FUNCTION_BLOCK E_SH_BYTE (* Sample-and-Hold for BOOL *)
  (* Standard: 61499-2 *)
  (* Version 1.0, 2024-02-23, franz *)
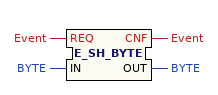
  EVENT_INPUT
    REQ; (* Normal Execution Request *)
  END_EVENT
  EVENT_OUTPUT
    CNF; (* Execution Confirmation *)
  END_EVENT
  VAR_INPUT
    IN : BYTE; (* Sample *)
  END_VAR
  VAR_OUTPUT
    OUT : BYTE; (* Hold *)
  END_VAR
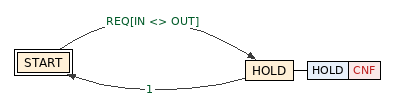
  EC_STATES
    START; (* Initial State *)
    HOLD : HOLD -> CNF;
  END_STATES
  EC_TRANSITIONS
    START TO HOLD := REQ[IN <> OUT];
    HOLD TO START := 1;
  END_TRANSITIONS
  ALGORITHM HOLD IN ST:
OUT := IN;
  END_ALGORITHM
END_FUNCTION_BLOCK
